VAR_GLOBAL

//Terminal EL1008
	DI1			AT%I*		:	BOOL;
	DI2			AT%I*		:	BOOL;
	DI3			AT%I*		:	BOOL;
	DI4			AT%I*		:	BOOL;
	DI5			AT%I*		:	BOOL;
	DI6			AT%I*		:	BOOL;
	DI7			AT%I*		:	BOOL;
	DI8			AT%I*		:	BOOL;
	
	SpindleEnable 				AT%Q*		:	BOOL;
	CoolingEnable				AT%Q*		:	BOOL; 
	
	ProximitySensorX			AT%I*		:	BOOL;
	ProximitySensorY			AT%I*		:	BOOL;
	ProximitySensorZ			AT%I*		:	BOOL;
	
	PistonSensorCutY 			AT%I*		:	BOOL;
	PistonSensorCutX			AT%I*		:	BOOL;
	
	PistonValveCutY				AT%Q*		:	BOOL;
	PistonValceCutX				AT%Q*		:	BOOL;	

END_VAR

(* stored: Version 1.1.0.1, ProductVersion 3.1.4024.15
   GVL IO: Id {28fb6f3d-0143-40a3-8031-ba6ef6dfc5ef} *)
